Staubli VAL3: remErrTimeout.pgx

program remErrTimeout(num& nTime[] (dimensions=1), string& sReturn[] (dimensions=1))
begin
  // Error raised when a command times out
  //
  logMsg("call remErrTimeout")
  sReturn="ERROR 401"
  sReturn=sReturn+": Timeout of cmd after "
  sReturn=sReturn+toString("",nTime)+" seconds."
  putln(sReturn)
  logMsg(sReturn)
end
